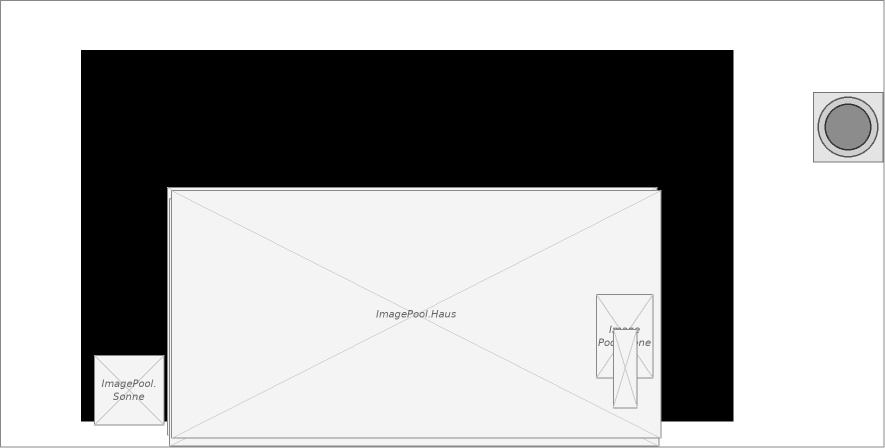
VISUALIZATION Haus  // 885x448
    Rectangle (81,50 652x371)
    Rectangle (81,50 652x371), colour variable: L_Background2
        p2167032090: L_Background2
    Image (167,187 490x248), invisible if: NOT L_Licht, image: ImagePool.Dunkel
    Image (169,198 490x248), invisible if: L_Licht, image: ImagePool.Licht
    Image (171,190 490x248), image: ImagePool.Haus
    PushSwitch (813,92 70x70), variable: L_Licht, behaviour: TOGGLE, style: Switch-PushSwitch-Gray
    Image (596,294 57x84), image: ImagePool.Krone
        p2858320360: L_Baum
    Image (613,329 24x79), image: ImagePool.Stamm
    Image (94,355 70x70), image: ImagePool.Sonne
        p2858320360: L_Sonnenstand
        p84334746: L_Sonne
END_VISUALIZATION

(* stored: Version 1.1.0.1, ProductVersion 3.1.4018.5
   Visu Haus: Id {3a34ba57-b0ad-46e3-811d-5feae23b576c} *)
